(* 17 Feb Practise Task *)

PROGRAM main
VAR
	Output : bool;
	InputA : bool;
	InputB : bool;
END_VAR

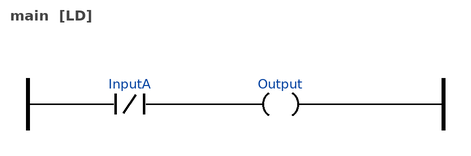
(* LD diagram, written out as Structured Text *)
Output := NOT InputA;
END_PROGRAM
